FUNCTION_BLOCK ExceptionHandling EXTENDS System IMPLEMENTS I_ExceptionHandling

VAR_OUTPUT
END_VAR
VAR
	{attribute 'hide'} 
	uiExceptionCounter : UINT := 0;
	uiPresentExceptions : UINT := 0;
	aExceptions : ARRAY[1..cMaxNumExceptions] OF ST_Exception;
	
	
	
END_VAR

VAR CONSTANT
	cMaxNumExceptions : UINT := 200;
	aEmptyExceptions : ARRAY[1..cMaxNumExceptions] OF ST_Exception;
END_VAR

SUPER^();

aExceptions := aEmptyExceptions;

uiExceptionCounter := 0;
uiPresentExceptions := 0;


METHOD BuildException : ST_Exception
VAR_INPUT
	eException	: E_Exception;
END_VAR
BuildException.eException := eException;
BuildException.eExceptionOrigin := getExceptionOrigin;
BuildException.sTimestamp := SYSTEMTIME_TO_STRING(fbTime.systemTime);
END_METHOD


METHOD Catch : BOOL
VAR_INPUT
	eException : E_Exception;
	eExceptionOrigin : E_Origin;
END_VAR

VAR

	i,k : UINT;
	stEmptyException : ST_Exception;
END_VAR
IF ExceptionAvailable()
THEN
	
	FOR i:= 1 TO uiExceptionCounter 
	DO
		//Search for exception
		IF aExceptions[i].eException = eException 
		AND_THEN aExceptions[i].eExceptionOrigin = eExceptionOrigin
		THEN
			//If found delete it from the array and adjust it
			Catch := TRUE;
			FOR k:= i TO uiExceptionCounter-1
			DO
				aExceptions[k] := aExceptions[k+1];
			END_FOR
			aExceptions[k+1] := stEmptyException;
			uiExceptionCounter := uiExceptionCounter - 1;
		END_IF  
	END_FOR

END_IF
END_METHOD

METHOD ExceptionAvailable : BOOL
ExceptionAvailable := uiExceptionCounter > 0;
END_METHOD

METHOD ForwardToNextLevel : BOOL
VAR_INPUT
	sender	: I_ExceptionHandling;
END_VAR
WHILE sender.ExceptionAvailable()
DO

	//Report to next level
	Throw(sender.getException);
	
END_WHILE
END_METHOD

METHOD GenericCatch : BOOL
VAR_INPUT
	eException	: E_Exception;
END_VAR
VAR
	i,k : UINT;
	stEmptyException : ST_Exception;
END_VAR
IF ExceptionAvailable()
THEN
	
	FOR i:= 1 TO uiExceptionCounter 
	DO
		//Search for exception
		IF aExceptions[i].eException = eException 
		THEN
			//If found delete it from the array and adjust it
			GenericCatch := TRUE;
			FOR k:= i TO uiExceptionCounter-1
			DO
				aExceptions[k] := aExceptions[k+1];
			END_FOR
			aExceptions[k+1] := stEmptyException;
			uiExceptionCounter := uiExceptionCounter - 1;
		END_IF  
	END_FOR

END_IF
END_METHOD

PROPERTY getException : ST_Exception
GET
IF ExceptionAvailable()
THEN
	getException := aExceptions[uiExceptionCounter];
	uiExceptionCounter := uiExceptionCounter - 1;
END_IF
END_GET
END_PROPERTY

PROPERTY getExceptionOrigin : E_Origin
GET
getExceptionOrigin := eOrigin;
END_GET
END_PROPERTY

METHOD Throw : BOOL
VAR_INPUT
	stException	: ST_Exception;
END_VAR
IF uiExceptionCounter <= cMaxNumExceptions
THEN
	uiExceptionCounter := uiExceptionCounter + 1;
	aExceptions[uiExceptionCounter] := stException;
	Throw := TRUE;
ELSE
	Throw := FALSE;
END_IF

uiPresentExceptions := uiExceptionCounter;
END_METHOD

END_FUNCTION_BLOCK

(* stored: Version 1.1.0.1, ProductVersion 3.1.4024.0
   POU ExceptionHandling: Id {6144b9ce-50bd-48d4-aa03-b6d39b8bbd11}, SpecialFunc None
   Method BuildException: Id {8efa5d74-d86d-4609-9105-696c907c4c69}
   Method Catch: Id {f9c63e61-7c30-4248-abfe-75c8e7452dd9}
   Method ExceptionAvailable: Id {b6619a72-f620-402d-8fc9-3f6300ec9a52}
   Method ForwardToNextLevel: Id {8630296e-c096-4a32-a199-6651c4c66622}
   Method GenericCatch: Id {8ce9b354-b72c-40fe-98ca-2e710962057e}
   Property getException: Id {be4c3491-9c15-48db-b0ce-03e8b0144da3}
   Get Get: Id {de30387b-0ad7-4f37-ac88-b30cb2da078b}
   Property getExceptionOrigin: Id {a314e47e-e18b-43e5-9b3f-13b39d10e3bc}
   Get Get: Id {ffd1d67d-ce26-452d-ae0e-5b04e35218bf}
   Method Throw: Id {6b6b8137-7798-4b20-b9a8-8c0ae3240d29} *)
